FUNCTION_BLOCK ABSTRACT ErrorManagerBase IMPLEMENTS IService
VAR_INPUT
END_VAR
VAR_OUTPUT
END_VAR
VAR
END_VAR

METHOD ABSTRACT AddMessage : BOOL
VAR_INPUT
	i_alarmId: UINT;
	i_active: BOOL;
	//i_acknowledged: BOOL;
	//i_confirmed: BOOL;
	i_severity: ESeverity;
	//i_retain: BOOL;
	i_instanceName: STRING;
	i_detailText: STRING := '';
END_VAR
END_METHOD

END_FUNCTION_BLOCK

(* stored: Version 1.1.0.1
   POU ErrorManagerBase: Id {860a830d-6c3c-4067-a206-91acd33451cb}, SpecialFunc None
   Method AddMessage: Id {7301fa91-c534-49c9-9e6b-860921dcdd0d} *)
